{attribute 'qualified_only'}
TYPE EL3433Index :
(	
	listStart	:= 3,
	ApparentPower:=3,
	Q,
	Energy,
	PF,
	Frequency,
	EnergyNegative,
	PhaseAngle,
	P1,
	S1,
	Q1,
	EnergyPositive,
	EnergyPositiveSaved,
	EnergySaved,
	EnergyNegativeSaved,
	FrequencyAvgRes,
	FrequencyHiRes,
	HeldFrequency,
	HeldFrequencyAvgRes,
	HeldFrequencyHiRes,
	listEnd := HeldFrequencyHiRes
);
END_TYPE

(* stored: Version 1.1.0.1, ProductVersion 3.1.4022.9
   DUT EL3433Index: Id {9974ad63-0f4c-4436-9c32-fd27fc1e6895} *)
